// TIA Portal V19 export
TYPE "LEXCHANGETRAY_typeSr1000ProfinetTelegram"
// stored: Access Published
   STRUCT
      in : "LEXCHANGETRAY_typeSr1000ProfinetTelegram_in";
      out : "LEXCHANGETRAY_typeSr1000ProfinetTelegram_out";
   END_STRUCT;
END_TYPE
